FUNCTION_BLOCK "AgainBullshit"
{ S7_Optimized_Access := 'TRUE' }
VERSION : 0.1
   VAR
      Auch : "Anwenderdatentyp_1";
      Und : "Anwenderdatentyp_1";
   END_VAR


BEGIN
	(* 4th edit *)
	(* 5th edit *)
	(* 6th edit *)
END_FUNCTION_BLOCK

